FUNCTION_BLOCK plant
  (* Standard: 61499-2 *)
  (* Version 0.1, 2015-00-13, Th?o, PC_THEO *)
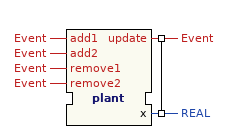
  EVENT_INPUT
    add1;
    add2;
    remove1;
    remove2;
  END_EVENT
  EVENT_OUTPUT
    update WITH x;
  END_EVENT
  VAR_OUTPUT
    x : REAL;
  END_VAR
  VAR
    d : REAL;
    k : INT;
    C1x : REAL;
  END_VAR
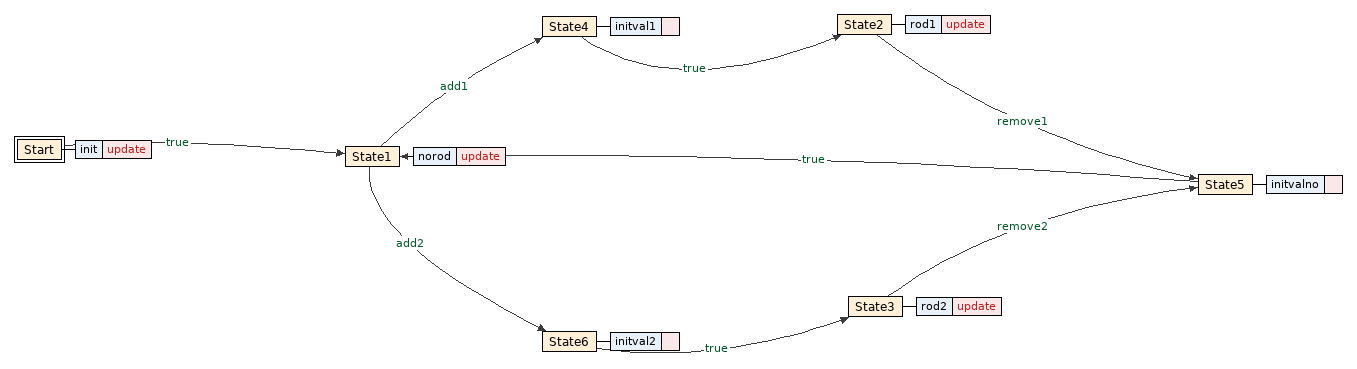
  EC_STATES
    Start : init -> update;
    State1 : norod -> update;
    State2 : rod1 -> update;
    State3 : rod2 -> update;
    State4 : initval1;
    State5 : initvalno;
    State6 : initval2;
  END_STATES
  EC_TRANSITIONS
    Start TO State1 := true;
    State1 TO State6 := add2;
    State1 TO State4 := add1;
    State2 TO State5 := remove1;
    State3 TO State5 := remove2;
    State4 TO State2 := true;
    State5 TO State1 := true;
    State6 TO State3 := true;
  END_TRANSITIONS
  ALGORITHM init IN C:
me->x=510;
me->d=0.01;
me->k=0;
me->C1x=10;
  END_ALGORITHM
  ALGORITHM norod IN C:
//me->x=me->C1x*exp(0.1*me->d*me->k) + 500.0;
me->x=550;
me->k++;
printf("No Rod, Temperature : %f\n",me->x);
  END_ALGORITHM
  ALGORITHM rod1 IN C:
//me->x = me->C1x*exp(0.1*me->d*me->k) + 560.0;
me->x=510;
me->k++;
printf("Rod1, Temperature : %f\n",me->x);
  END_ALGORITHM
  ALGORITHM rod2 IN C:
//me->x = me->C1x*exp(0.1*me->d*me->k) + 600.0;
me->x=510;
me->k++;
printf("Rod2, Temperature : %f\n",me->x);
  END_ALGORITHM
  ALGORITHM initvalno IN C:
me->k=0;
me->C1x=me->x-500;
  END_ALGORITHM
  ALGORITHM initval1 IN C:
me->k=0;
me->C1x=me->x-560;
  END_ALGORITHM
  ALGORITHM initval2 IN C:
me->k=0;
me->C1x=me->x-600;
  END_ALGORITHM
END_FUNCTION_BLOCK
